Fanuc KAREL source: kd00033.KL

-- PROVISIONAL review KL for V770-1; original PC SHA256 535c64ee993c859f58c9d8de08852c505151b180e0eb8d4cd3399d2dd838febb
-- Incomplete behavior may be omitted. Consult companion uncertainty JSON. Do not deploy.
PROGRAM KD00033
%NOLOCKGROUP
VAR
  I : INTEGER
  J : INTEGER
  B : BOOLEAN
  R : REAL
  S : STRING[80]
BEGIN
  -- UNRESOLVED_PC offsets 5-24; opcodes 9D,81,18,9D,1B,9D,12,22,9D,13,04
  -- UNRESOLVED_PC offsets 29-33; opcodes 7F
END KD00033
